// TIA Portal V20 export
TYPE "LKinCtrl_typeCOffCmdOutInternal"
   STRUCT
      cmdType : Int := -1;   // 1: MoveLinAbs; 2: MoveLinRel; 3: MoveCircAbs; 4: MoveCircRel; 5: MoveDirectAbs; 6: MoveDirectRel; 10: TrackConveyorBelt; 100: WaitTime; 40/41/42: ContourOffset; 0: FlagOnlyCmd; -1: End of List
      endPoint : "LKinCtrl_typeCOff3DPoint";   // end point of command
      circleMode : DInt;   // 0: auxPoint defines point on circle line; 1: auxPoint defines circle center; 2: radius and endPoint define circle segment
      circleCenterPoint : "LKinCtrl_typeCOff3DPoint";   // center point of circle
      circleIntermediatePoint : "LKinCtrl_typeCOff3DPoint";   // intermediate point of circle
      transitionParameter1 : LReal;   // transition parameter
      endPointOrthShifted : "LKinCtrl_typeCOff3DPoint";   // orthogonal shifted end point of command
      endPointOrthTangShifted : "LKinCtrl_typeCOff3DPoint";   // orthogonal and tangential shifted end point of command
      startPointOrthShifted : "LKinCtrl_typeCOff3DPoint";   // orthogonal shifted end point of command
      startPointOrthTangShifted : "LKinCtrl_typeCOff3DPoint";   // orthogonal and tangential shifted end point of command
      circleRadius : LReal;   // circle radius
      circleAngle : LReal;   // circle angle
      orthogonalUnitVecEnd : "LKinCtrl_typeCOff3DPoint";   // orthogonal unit vector end
      tangentialUnitVecEnd : "LKinCtrl_typeCOff3DPoint";   // tangential unit vector end
      orthogonalShiftEnd : "LKinCtrl_typeCOff3DPoint";   // orthogonal shift end
      tangentiaShiftEnd : "LKinCtrl_typeCOff3DPoint";   // tangential shift end
      orthogonalUnitVecStart : "LKinCtrl_typeCOff3DPoint";   // orthogonal unit vector start
      tangentialUnitVecStart : "LKinCtrl_typeCOff3DPoint";   // tangential unit vector start
      orthogonalShiftStart : "LKinCtrl_typeCOff3DPoint";   // orthogonal shift start
      tangentiaShiftStart : "LKinCtrl_typeCOff3DPoint";   // tangential shift start
      orthogonalUnitVecIntermediate : "LKinCtrl_typeCOff3DPoint";   // orthogonal unit vector intermediate
      tangentialUnitVecIntermediate : "LKinCtrl_typeCOff3DPoint";   // tangential unit vector intermediate
      orthogonalShiftIntermediate : "LKinCtrl_typeCOff3DPoint";   // orthogonal shift intermediate
   END_STRUCT;
END_TYPE
